PROGRAM WaterFlowControl
VAR
END_VAR

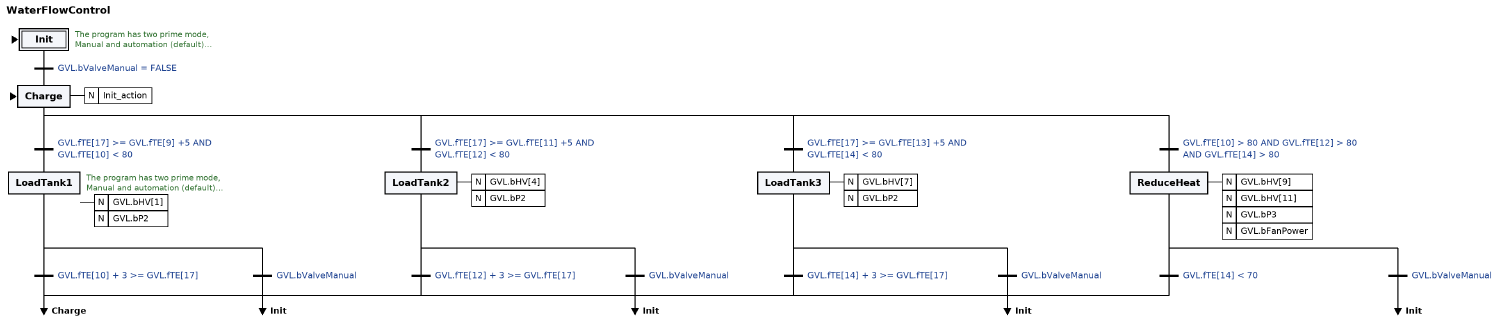
// The program has two prime mode, Manual and automation (default). Manual mode counteracts the whole program so that you can control flows as you want. In automation mode, if boiler water temperature is at least 5 degree greater than tank water's, and tank water is lower than 80 degree; valve and pump will be turned on to load water to tank. If more than one tank meet the requirements, the loading process order will be 1,2,3. There's always one tank being loaded at a time. If 3 tanks have above 80 degree temperature, pump 3 and corresponding valves will be opened to unload the heat. If tank temperature is greater than boiler's, loading will stop in order to avoid heat loss. Consider having most critical condition/function on the most left branches, because in alternative branches, the order is from left to right.
INITIAL_STEP Init:
END_STEP
TRANSITION FROM Init TO Charge
    := GVL.bValveManual = FALSE;
END_TRANSITION
STEP Charge:
    Init_action(N);
END_STEP
TRANSITION FROM Charge TO LoadTank1
    := GVL.fTE[17] >= GVL.fTE[9] +5 AND GVL.fTE[10] < 80;
END_TRANSITION
// The program has two prime mode, Manual and automation (default). Manual mode counteracts the whole program so that you can control flows as you want. In automation mode, if boiler water temperature is at least 5 degree greater than tank water's, and tank water is lower than 80 degree; valve and pump will be turned on to load water to tank. If more than one tank meet the requirements, the loading process order will be 1,2,3. There's always one tank being loaded at a time. If 3 tanks have above 80 degree temperature, pump 3 and corresponding valves will be opened to unload the heat. If tank temperature is greater than boiler's, loading will stop in order to avoid heat loss. Consider having most critical condition/function on the most left branches, because in alternative branches, the order is from left to right.
STEP LoadTank1:
    GVL.bHV[1](N);
    GVL.bP2(N);
END_STEP
TRANSITION FROM LoadTank1 TO Charge
    := GVL.fTE[10] + 3 >= GVL.fTE[17];
END_TRANSITION
TRANSITION FROM LoadTank1 TO Init
    := GVL.bValveManual;
END_TRANSITION
TRANSITION FROM Charge TO LoadTank2
    := GVL.fTE[17] >= GVL.fTE[11] +5 AND GVL.fTE[12] < 80;
END_TRANSITION
STEP LoadTank2:
    GVL.bHV[4](N);
    GVL.bP2(N);
END_STEP
TRANSITION FROM LoadTank2 TO Charge
    := GVL.fTE[12] + 3 >= GVL.fTE[17];
END_TRANSITION
TRANSITION FROM LoadTank2 TO Init
    := GVL.bValveManual;
END_TRANSITION
TRANSITION FROM Charge TO LoadTank3
    := GVL.fTE[17] >= GVL.fTE[13] +5 AND GVL.fTE[14] < 80;
END_TRANSITION
STEP LoadTank3:
    GVL.bHV[7](N);
    GVL.bP2(N);
END_STEP
TRANSITION FROM LoadTank3 TO Charge
    := GVL.fTE[14] + 3 >= GVL.fTE[17];
END_TRANSITION
TRANSITION FROM LoadTank3 TO Init
    := GVL.bValveManual;
END_TRANSITION
TRANSITION FROM Charge TO ReduceHeat
    := GVL.fTE[10] > 80 AND GVL.fTE[12] > 80 AND GVL.fTE[14] > 80;
END_TRANSITION
STEP ReduceHeat:
    GVL.bHV[9](N);
    GVL.bHV[11](N);
    GVL.bP3(N);
    GVL.bFanPower(N);
END_STEP
TRANSITION FROM ReduceHeat TO Charge
    := GVL.fTE[14] < 70;
END_TRANSITION
TRANSITION FROM ReduceHeat TO Init
    := GVL.bValveManual;
END_TRANSITION

ACTION Init_action:
(*GVL.bHV[1] := FALSE;
GVL.bHV[2] := FALSE;
GVL.bHV[3] := FALSE;
GVL.bHV[4] := FALSE;
GVL.bHV[5] := FALSE;
GVL.bHV[6] := FALSE;
GVL.bHV[7] := FALSE;
GVL.bHV[8] := FALSE;
GVL.bHV[9] := FALSE;
GVL.bHV[10] := FALSE;*)
GVL.bP2 := FALSE;
GVL.bP3 := FALSE;
END_ACTION

END_PROGRAM

(* stored: Version 1.1.0.1, ProductVersion 3.1.4022.18
   POU WaterFlowControl: Id {dd4a8b65-c70f-4ce7-a7a1-31ab5aeb7556}, SpecialFunc None
   Action Init_action: Id {757bc54f-6647-490d-882a-37e9eff902bd} *)
